// Mitsubishi GX Works2 project: 機電整合丙級第四題-ST   PLC: FX3U/FX3UC

// task Task_01 (event TRUE, interval 0, priority 31): POU_01

PROGRAM POU_01
VAR
  wProgramStep : INT;
  bM17 : BOOL;
  bM24 : BOOL;
  bM44 : BOOL;
  bM123 : BOOL;
  tdT123 : TON;
  tdT24 : TON;
  wCountOf2 : INT;
  bMetal : BOOL;
  tdT22 : TON;
  tdT31 : TON;
  tdT35 : TON;
  bM12 : BOOL;
  tdT23 : TON;
  tdT125 : TON;
END_VAR
(* 機電整合丙級術科第四題
   Author: Steven Luo
   Date: 2018/09/26
*)

IF M8002 OR NOT X17 THEN
	wProgramStep := 0;
	ZRST(TRUE, Y0, Y17);
	bM17 := FALSE;
	bM123 := FALSE;
END_IF;

IF NOT X17 THEN (* 按下急停 *)
	bM17 := TRUE;
END_IF;

IF X17 AND bM17 THEN (* 放開急停，等待復歸 *)
	wProgramStep := 122;
END_IF;

IF M8002 THEN
	wProgramStep := 21;
END_IF;

IF bM123 THEN
	IF M8013 THEN
		SET(TRUE, Y16); (* 黃燈閃爍 *)
	ELSE
		RST(TRUE, Y16);
	END_IF;
	tdT123(IN := TRUE, PT := T#3s); (* 計時三秒 *)
ELSE
	RST(TRUE, Y16);
END_IF;

IF X12 THEN
	bM12 := TRUE;
END_IF;

CASE wProgramStep OF
	21:
		IF X1 AND X3 AND X4 AND (*X6 AND*) NOT X11 THEN
			SET(TRUE, Y17); (* 待機，綠燈亮、紅燈滅 *)
			RST(TRUE, Y15);
			bM12 := FALSE;
			bM123 := FALSE;
			bM24 := FALSE;
			bM44 := FALSE;
		END_IF;
		IF X13 AND X17 AND X10 AND X16 THEN (* 工作模式、按下啟動鈕 *)
			tdT123(IN := FALSE);
			tdT22(IN := FALSE);
			SET(TRUE, Y15); (* 紅燈亮、綠燈滅 *)
			RST(TRUE, Y17);
			wProgramStep := 22;
		END_IF;
	22:
		IF X10 THEN (* 有料 *)
			wCountOf2 := 0;
			IF X7 THEN (* 鋁料 *)
				bMetal:= TRUE;
			ELSE (* 塑膠料 *)
				bMetal := FALSE;
			END_IF;
			tdT22(IN := TRUE, PT := T#2s); (* 計時二秒 *)
			IF tdT22.Q AND NOT X11 THEN
				tdT23(IN := FALSE);
				wProgramStep := 23;
			END_IF;
		END_IF;
	23:
		IF X1 AND X3 AND X4 THEN
			SET(TRUE, Y6); (*分度盤轉 *)
			tdT23(IN := TRUE, PT := T#200ms);
			IF tdT23.Q AND X6 THEN
				wCountOf2 := wCountOf2 + 1;
				IF wCountOf2 = 1 THEN (* 90度 *)
					IF NOT bMetal OR NOT X14 THEN (* 蓋印 *)
						tdT24(IN := FALSE);
						wProgramStep := 24;
					ELSE (* 指定功能、鋁料 *)
						tdT31(IN := FALSE);
						wProgramStep := 31;
					END_IF;
				ELSIF wCountOf2 = 2 THEN (* 180度 *)
					IF bMetal THEN (* 指定功能、鋁料、鑽孔 *)
						tdT35(IN := FALSE);
						wProgramStep := 34;
					ELSE (* 塑料 *)
						tdT31(IN := FALSE);
						wProgramStep := 31;
					END_IF;
				ELSIF wCountOf2 = 3 THEN (* 270度 *)
					wProgramStep := 25; (* 出料 *)
				END_IF;
			END_IF;
		END_IF;
	24:
		RST(TRUE, Y6); (* 分度盤停止 *)
		SET(TRUE, Y0); (* 蓋印缸下降 *)
		IF X0 THEN
			tdT24(IN := TRUE, PT := T#1s);
			IF tdT24.Q THEN
				RST(TRUE, Y0); (* 蓋印缸上升 *)
				tdT23(IN := FALSE);
				wProgramStep := 23;
			END_IF;
		END_IF;
	25:
		RST(TRUE, Y6); (* 分度盤停止 *)
		SET(TRUE, Y16); (* 黃燈亮、手動出料 *)
		IF NOT X11 THEN
			RST(TRUE, Y16);
			IF X15 THEN (* 連續循環 *)
				IF bM12 THEN (* 按下停止鈕 *)
					wProgramStep := 21;
				ELSE
					tdT22(IN := FALSE);
					wProgramStep := 22;
				END_IF;
			ELSE (* 單一循環、指定功能 *)
				wProgramStep := 21;
			END_IF;
		END_IF;
	31:
		tdT31(IN := TRUE, PT := T#1s); (* 延遲一秒 *)
		IF tdT31.Q THEN
			tdT23(IN := FALSE);
			wprogramStep := 23;
		END_IF;
	34:
		RST(TRUE, Y6); (* 分度盤停止 *)
		SET(TRUE, Y5); (* 夾料缸前進 *)
		IF X5 THEN
			RST(TRUE, Y5);
			wProgramStep := 35;
		END_IF;
	35:
		SET(TRUE, Y7); (* 鑽孔馬達旋轉 *)
		SET(TRUE, Y2); (* 鑽孔缸下降 *)
		IF X2 THEN
			RST(TRUE, Y2);
			tdT35(IN := TRUE, PT := T#1s);
			IF tdT35.Q THEN
				wProgramStep := 36;
			END_IF;
		END_IF;
	36:
		SET(TRUE, Y3); (* 鑽孔缸上升 *)
		IF X3 THEN
			RST(TRUE, Y3);
			wProgramStep := 37;
		END_IF;
	37:
		RST(TRUE, Y7); (* 鑽孔馬達停止 *)
		SET(TRUE, Y4); (* 夾料缸後退 *)
		IF X4 THEN
			RST(TRUE, Y4);
			tdT23(IN := FALSE);
			wProgramStep := 23; (*分度盤轉90度 *)
		END_IF;
	122:
		IF NOT X13 AND X16 THEN (* 復歸模式、按下復歸開關 *)
			bM17 := FALSE;
			wProgramStep := 123;
		END_IF;
	123:
		bM123 := TRUE;
		SET(TRUE, Y3); (* 鑽孔缸上升 *)
		IF X3 THEN
			RST(TRUE, Y3);
			wProgramStep := 124;
		END_IF;
	124:
		SET(TRUE, Y4); (* 夾料缸後退 *)
		IF X4 THEN
			RST(TRUE, Y4);
			tdT125(IN := FALSE);
			wProgramStep := 125;
		END_IF;
	125:
		SET(TRUE, Y6); (*分度盤轉90度 *)
		tdT125(IN := TRUE, PT := T#200ms);
		IF tdT125.Q AND X6 THEN
			RST(TRUE, Y6); (* 分度盤停止 *)
			IF tdT123.Q THEN
				bM123 := FALSE;
				wProgramStep := 21;
			END_IF;
		END_IF;
	ELSE
	;
END_CASE;
END_PROGRAM
